PROGRAM MAIN
VAR
	SmartHome : SmartHomeOfUncleSasha;
	
	Home : REFERENCE TO SHLib.SmartHome<5>; 
END_VAR

IF NOT __ISVALIDREF(Home) THEN	
	Home REF= SmartHome; 
END_IF

Home.Execute();

END_PROGRAM

(* stored: Version 1.1.0.1
   POU MAIN: Id {23cba3fb-552e-4b11-b57f-a311785ea557}, SpecialFunc None *)
